// TwinCAT 3 PLC project ShapeMonitor
// ProgramVersion: 3.1.4023.0
// CompilerDefines: VISU_USEWSTRING
// libraries:
//   Tc2_EtherCAT, * (Beckhoff Automation GmbH)
//   Tc2_MDP, * (Beckhoff Automation GmbH)
//   Tc2_ModbusSrv, * (Beckhoff Automation GmbH)
//   Tc2_Standard, * (Beckhoff Automation GmbH)
//   Tc2_System, * (Beckhoff Automation GmbH)
//   Tc2_Utilities, * (Beckhoff Automation GmbH)
//   Tc3_IotBase, * (Beckhoff Automation GmbH)
//   Tc3_IPCDiag, * (Beckhoff Automation GmbH)
//   Tc3_JsonXml, * (Beckhoff Automation GmbH)
//   Tc3_Module, * (Beckhoff Automation GmbH)
//   BASIC,3.31,OSCAT
//   Tc2_SUPS,3.3.8.0,Beckhoff Automation GmbH
//   VisuSymbols,3.5.10.0,System
// project tree:
//   / GlobalTextList.TcGTLO, PlcTask_10ms.TcTTO
//   GVLs/ constGVL.TcGVL, GVL.TcGVL, GVL_outputs.TcGVL
//   HMI/ VisualizationManager.TcVMO (not stored)
//   POUs/FB/ ShapeMonitor.TcPOU
//   POUs/PRG/ Monitoring.TcPOU, Main_T10ms.TcPOU
//   Simulation/ Simulation.TcPOU
// real-time tasks:
//   TASK PlcTask_10ms: cycle T#10ms, priority 20, ADS port 350

CONFIGURATION ShapeMonitor
    RESOURCE PLC ON TwinCAT3
        TASK PlcTask_10ms(INTERVAL := T#10ms, PRIORITY := 20);
        PROGRAM Main_T10ms WITH PlcTask_10ms : Main_T10ms;
    END_RESOURCE
END_CONFIGURATION

// ---- GVLs/constGVL.TcGVL
{attribute 'qualified_only'}
VAR_GLOBAL
	
	//ipHostAddress	: STRING		:= '192.168.1.170';
	ipHostAddress	: STRING		:= '10.1.226.41';
	
	HostPort		: UINT			:= 1883;
	UserName		: STRING		:= 'mqttbroker';
	//UserPassword	: STRING		:= 'LoopEdge.123';
	UserPassword	: STRING		:= 'PLWRO@mqtt';
	
	WorkCenter 		: STRING(30)	:= 'PLPSDWB1';
	LineName 		: STRING(30)	:= 'PSD_WB';
	MachineName01 	: STRING(30)	:= 'WB1';
	MachineTopic_Status01 : STRING	:= 'MachineStatus';
	
	// Config for InfluxDB
	//ActuatorOperTimes_InfluxMeas 	: STRING(50) := 'ActuatorOperTimes';
	VibAccelAnomaly_InfluxMeas 		: STRING(50) := 'VibAccelAnalytics';
	VibVeloAnomaly_InfluxMeas 		: STRING(50) := 'VibVeloAnalytics';
	MachineState_InfluxMeas 		: STRING(50) := 'MachineStatus';
	EdgeDiag_InfluxMeas 			: STRING(50) := 'EdgeGateway';
	FlowSensor_InfluxMeas 			: STRING(50) := 'FlowSensor';
	PressureSensor_InfluxMeas		: STRING(50) := 'PressureSensor';
	PositionSensor_InfluxMeas		: STRING(50) := 'PositionSensor';
	ShapeCorrelation_InfluxMeas		: STRING(50) := 'ShapeCorrelation';
	//TempHumidSensor_InfluxMeas 	: STRING(50) := 'TempHumidSensor';
	//ElectricalData_InfluxMeas		: STRING(50) := 'ElectricalMeasurement';
	
	BF1	:STRING			:= 'BF1';	// przepływ powietrza - zasilanie maszyny
	
	BP1	:STRING			:= 'BP1';	// cisnienie powietrza  - docisk rolek na reduktorem
	BP2	:STRING			:= 'BP2';	// cisnienie powietrza  - odwijanie drutu
	BP3	:STRING			:= 'BP3';	// cisnienie powietrza  - przy enkoderze
	
	// separate vibration sensors 
	BS1 			:STRING			:= 'BS1';		//	wibracje przy kole zębatym - napęd	
	BS2 			:STRING			:= 'BS2';		//	wibracje przy kole zębatym - na obudowie
	BS3				:STRING			:= 'BS3';		// wibracje przy AccuLathe
	
	BG01			:STRING			:='BG01';		// polożenie ciągle ramienia na odwijaku
	BG02			:STRING			:='BG02';		// połozenie binarne ramienia na odwijaku
	
END_VAR

VAR_GLOBAL CONSTANT
	// *******************Global Const ************************
	LeverArmShapeMaxNoSample: UINT := 200;
END_VAR

// ---- GVLs/GVL.TcGVL
{attribute 'qualified_only'}
VAR_GLOBAL
	
(********************* TimeStamp *********************)
	Unix_TimeStamp 			: ULINT;
	
(********************* Machine States *********************)
	AutoMode 				: BOOL;
	ManualMode 				: BOOL;
	MachineProducing		: BOOL;
	DoorGuardSts 			: BOOL;
	ESTOP_NOK				: BOOL;
	
	WireCutSignal			: BOOL;		// command for cutting wire 
	Robot_Error				: BOOL;
	HeatingErrorDepot3		: BOOL;		// heating error on depot 3 (corner)
	HeatingErrorDepot2		: BOOL;		// heating error on depot 2 (middle)
	RobotRunMode			: BOOL;
	WelderRunning			: BOOL;
	WelderReady				: BOOL;
	WelderHeatingOn			: BOOL;
	LifeBeat				: BOOL;		// life bit 1 sec.
	ConnectionOK			: BOOL;		// monitoring of LifeBeat
	FieldbusOK				: BOOL;		// EtherCat communication OK.
	


(**********************************************************)
	ProductOK: DINT;		// amount of finished OK product 
	ProductNOK:	DINT;		// amount of NOK product
	ProductCantNOK:	DINT;	// amount of NOK cant product 
	
	// Data from HMI (PS4800) at WB4
	DataHmi2TwinCat							: ARRAY[1..4] OF DINT;
	
END_VAR

// ---- GVLs/GVL_outputs.TcGVL
{attribute 'qualified_only'}
VAR_GLOBAL
	
	// Data to Allen Bradley over EtherNet/IP
	DataEthNetIP_OUTPUT_DINT0				AT%Q*: DINT;
	DataEthNetIP_OUTPUT_DINT1				AT%Q*: DINT;
END_VAR

// ---- POUs/PRG/Main_T10ms.TcPOU
PROGRAM Main_T10ms
VAR

END_VAR

Simulation();

Monitoring();

END_PROGRAM

// ---- Simulation/Simulation.TcPOU
PROGRAM Simulation
VAR
	BaseValues				:	ARRAY [0..BASE_SHAPE_SAMPLES_NO] OF REAL := [0.1, 0.2, 0.3, 0.5, 0.8, 0.9, 1.0, 1.05, 1.15, 1.25, 1.4, 1.6, 1.8, 2.0, 2.4, 2.8, 3.2, 3.7, 4.1, 4.7, 5.15, 5.6, 6.1, 6.5, 6.95, 7.3, 7.6, 7.9, 8.1, 8.3, 8.4, 3(8.5), 8.4, 8.2, 8.1, 8.0, 7.8, 7.7, 7.5, 7.3, 7.0, 6.98, 6.9, 6.85, 6.9, 6.87, 6.88, 6.85, 6.84, 6.83, 6.84, 6.82, 6.81, 6.82, 6.81, 6.83, 6.8, 6.75, 6.7, 6.65, 6.6, 6.55, 6.5, 6.45, 6.4, 6.35, 6.3, 6.25, 6.2, 6.1, 5.9, 5.8, 5.6, 5.5, 5.32, 5.25, 5.2, 5.0, 4.8, 4.6, 4.4, 4.1, 3.7, 3.4, 3.05, 2.8, 2.6, 2.4, 2.3, 2.1, 1.9, 1.7, 1.5, 1.3, 1.0, 0.7, 0.5, 0.3];
	ValueOffset				:	REAL;
	MeasuredValues			:	ARRAY [0..BASE_SHAPE_SAMPLES_NO] OF REAL;
	Idx						:	UINT;
	SimValue				:	DRAND();
	
	tp01					: 	TP;
	tp02					: 	TP;
	rtShapeStart			:	R_TRIG;
	ftShapeStop				:	F_TRIG;
	ShapeStarted			:	BOOL;
	MeasuredValue			:	REAL;
	SimEnable				:	BOOL;
END_VAR

VAR CONSTANT
	BASE_SHAPE_SAMPLES_NO	: 	UINT:=99;
END_VAR

tp01(IN:=SimEnable AND NOT tp02.Q , PT:=T#1000MS , Q=> , ET=> );
tp02(IN:=NOT tp01.Q , PT:=T#500MS , Q=> , ET=> );

rtShapeStart(CLK:=tp01.Q);
ftShapeStop(CLK:=tp01.Q);

IF rtShapeStart.Q THEN
	ShapeStarted := TRUE;
	Idx := 0;
END_IF

IF ftShapeStop.Q THEN
	ShapeStarted := FALSE;
	MeasuredValue := 0;
END_IF


IF ShapeStarted THEN
	SimValue(Seed:=2);
	ValueOffset := LREAL_TO_REAL(SimValue.Num) - 0.5;
	MeasuredValues[Idx] := BaseValues[Idx] + (0.1 * ValueOffset);
	MeasuredValue := MeasuredValues[Idx];
	Idx := Idx + 1;
	IF Idx > BASE_SHAPE_SAMPLES_NO THEN
		Idx := 0;
		MeasuredValue := 0;
	END_IF
END_IF


//FOR Idx:=0 TO BASE_SHAPE_SAMPLES_NO DO
//	SimValue(Seed:=2);
//	ValueOffset := LREAL_TO_REAL(SimValue.Num) - 0.5;
	
//	MeasuredValues[Idx] := BaseValues[Idx] + (0.2 * ValueOffset);
//END_FOR

END_PROGRAM

// ---- POUs/PRG/Monitoring.TcPOU
PROGRAM Monitoring
VAR	

END_VAR

VAR RETAIN PERSISTENT
	ShapeMonitor01					:	ShapeMonitor;
END_VAR

ShapeMonitor01(
    AnalogIn := Simulation.MeasuredValue,
    TriggerSensor := Simulation.ShapeStarted,
    Enable := TRUE); // ShapeMonitor

END_PROGRAM

// ---- POUs/FB/ShapeMonitor.TcPOU
FUNCTION_BLOCK ShapeMonitor
VAR_INPUT
	AnalogIn											: REAL;
	TriggerSensor										: BOOL;
	Enable												: BOOL;
	Reset												: BOOL;							// reset algorithm
END_VAR
VAR_OUTPUT
	BaseInCalculation									: BOOL;							// base model during calculation
	BaseCompleted										: BOOL;							// model base calculation completed
	SumSquaredError										: REAL;							// SSE - sumed squared error
	Busy												: BOOL;							// shape evaluation in progress 
	Done												: BOOL;							// shape evaluated
END_VAR	

			
VAR
	rtTriggerSensor										: R_TRIG;						// detect rising edge of trigger sensor
	ftTriggerSensor										: F_TRIG;						// detect falling edge of trigger sensor
	rtReset												: R_TRIG;						// detect rising edge of reset signal
	
	State												: (IDLE, TRIGGER_STARTED, TRIGGER_STOPPED );		// state machine
	
	arrShapeSamples										: ARRAY [0..SAMPLES_IN_SHAPE] OF REAL;				// real-time analog samples catched at each PLC scan				
	IdxMeasureSample		   							: UINT;												// index of real-time measured sample 
	
	arrBaseSamples										: ARRAY[0..SHAPES_IN_BASE] OF ARRAY [0..SAMPLES_IN_SHAPE] OF REAL;	// collected real-time signal shapes in base shapes 
	arrNoSamplesInBaseShape								: ARRAY[0..SHAPES_IN_BASE] OF UINT;									// number of samples in each base shape
	arrBase												: ARRAY[0..SAMPLES_IN_SHAPE] OF REAL;								// averaged base shapes array 
	
	arrResult											: ARRAY [0..SAMPLES_IN_SHAPE] OF REAL;								// array with squared diff. between base and incoming new shape
	
	NoBaseShapes										: UINT;																// number of collected shapes in 'base'
	IdxBaseShape										: UINT;																// idx for shape iteration
	IdxSample											: UINT;																// idx for sample iteration
																	
	MaxBaseLength										: UINT;																// max length of shapes in base model
	SampleLength										: UINT;																// length(num of samples) of evaluated shape
	Total												: REAL;																// temporary var
																
END_VAR


VAR CONSTANT
	SHAPES_IN_BASE										: UINT := 10;				// number of shape samples in base
	SAMPLES_IN_SHAPE									: UINT:= 199;				// max number of samples in one shape
END_VAR

// detect rising trigger from reset input	
rtReset(CLK:=Reset , Q=> );	
IF rtReset.Q THEN 
	resetAlgorithm();
END_IF;


IF ENABLE THEN
	
	// detect rising edge of trigger sensor	
	rtTriggerSensor(CLK:=TriggerSensor , Q=> );
	
	// detect falling edge of trigger sensor
	ftTriggerSensor(CLK:=TriggerSensor , Q=> );
	
	CASE State OF
	IDLE:
		// clear array with measured data samples
		MEMSET(ADR(arrShapeSamples), 0, SIZEOF(arrShapeSamples));
		IdxMeasureSample 		:= 0;
		Busy					:= FALSE;	
		Done 					:= FALSE;
		
		IF rtTriggerSensor.Q THEN
			// WatchDog_State_ton.IN := TRUE; //sequence watchdog
			State := TRIGGER_STARTED;
		END_IF
		
	TRIGGER_STARTED:
	// trigger sensor entered start position
		Busy				:= TRUE;	
		Done 				:= FALSE;
		
		// fill the array with incoming measured data
		arrShapeSamples[IdxMeasureSample] := AnalogIn;
		IdxMeasureSample := IdxMeasureSample + 1;
		
		// trigger sensor reached stop position OR max number of samples already collected	
		IF ftTriggerSensor.Q OR IdxMeasureSample > SAMPLES_IN_SHAPE  THEN
			State := TRIGGER_STOPPED;					
		END_IF
		
	TRIGGER_STOPPED:
	// trigger sensor left start position or max no of samples collected
		
		// collect shapes for 'Base' 
		IF NoBaseShapes < SHAPES_IN_BASE  THEN
			BaseInCalculation := TRUE;
			arrBaseSamples[NoBaseShapes] := arrShapeSamples;
			NoBaseShapes := NoBaseShapes + 1;
		
		// shapes for base already collected
		ELSE
			// base calculation not completed yet
			IF NOT BaseCompleted THEN
				
				// find max length of each shape in 'Base'
				FOR IdxBaseShape := 0 TO SHAPES_IN_BASE-1 BY 1 DO
					FOR idxSample := 0 TO SAMPLES_IN_SHAPE BY 1 DO
						IF arrBaseSamples[IdxBaseShape][idxSample] = 0 THEN
							arrNoSamplesInBaseShape[IdxBaseShape] := idxSample-1;
							EXIT;
						END_IF
					END_FOR
				END_FOR
				
				// find max length of all base shapes
				MaxBaseLength 	:= 	0;
				FOR IdxMeasureSample := 0 TO SHAPES_IN_BASE-1 BY 1 DO
					IF arrNoSamplesInBaseShape[IdxMeasureSample] > MaxBaseLength THEN 
						MaxBaseLength:= arrNoSamplesInBaseShape[IdxMeasureSample]; 
					END_IF
				END_FOR
				
				// equalize signal length for all collected base shapes (add last point)
				FOR IdxBaseShape := 0 TO SHAPES_IN_BASE-1 BY 1 DO
					IF arrNoSamplesInBaseShape[IdxBaseShape] <  MaxBaseLength THEN
						FOR IdxSample := arrNoSamplesInBaseShape[IdxBaseShape] TO MaxBaseLength BY 1 DO
							 arrBaseSamples[IdxBaseShape][IdxSample] := arrBaseSamples[IdxBaseShape][ arrNoSamplesInBaseShape[IdxBaseShape]];
						END_FOR
					END_IF
				END_FOR

				// calculate avarage of all samples in BaseSamples -> create one 'Base' array
				FOR IdxSample := 0 TO MaxBaseLength BY 1 DO
					Total := 0;
					FOR  IdxBaseShape := 0 TO SHAPES_IN_BASE-1 BY 1 DO
						Total := Total + arrBaseSamples[IdxBaseShape][IdxSample];
					END_FOR
					arrBase[IdxSample] := Total / (SHAPES_IN_BASE); 
				END_FOR
				
				BaseCompleted	:=	TRUE;
				
			ELSIF BaseCompleted AND
				// ensure that valid number of samples was collected 
				(UINT_TO_REAL(IdxMeasureSample) < 1.1 * UINT_TO_REAL(MaxBaseLength) AND
				 UINT_TO_REAL(IdxMeasureSample) > 0.9 * UINT_TO_REAL(MaxBaseLength) ) THEN
				 
				 BaseInCalculation := FALSE;
				 
				// find length of incoming shape
				FOR IdxSample := 0 TO SAMPLES_IN_SHAPE BY 1 DO
					IF arrShapeSamples[idxSample] = 0 THEN
						SampleLength := idxSample;
						// exit FOR loop when element with value 0 found 
						EXIT;
					END_IF
				END_FOR
				
				// adjust incoming shape length equal to base length by adding last value
				IF SampleLength < MaxBaseLength THEN
					FOR IdxSample := SampleLength TO MaxBaseLength BY 1 DO
						arrShapeSamples[IdxSample] := arrShapeSamples[SampleLength-1];
					END_FOR
				END_IF
				
				// calculate difference between base and measured shape => error and square error value
				FOR IdxSample := 0 TO MaxBaseLength BY 1 DO
					arrResult[idxSample] := LREAL_TO_REAL(EXPT((arrBase[idxSample] - arrShapeSamples[idxSample]),2)) ;
				END_FOR
				
				// calculate sum of squared errors (SSE)
				SumSquaredError := 0;
				FOR IdxSample := 0 TO MaxBaseLength BY 1 DO
					SumSquaredError := SumSquaredError + arrResult[idxSample];
				END_FOR
				
				
			// new samples number is outside of limits -> restart algorithm
			ELSIF BaseCompleted AND (UINT_TO_REAL(IdxMeasureSample) > 1.2 * UINT_TO_REAL(MaxBaseLength)) OR
				  (UINT_TO_REAL(IdxMeasureSample) < 0.8 * UINT_TO_REAL(MaxBaseLength)) THEN
				  // withdraw this shape because too many/too less samples collected
				  resetAlgorithm();
			END_IF
	
		END_IF
		
		
		Busy					:= FALSE;	
		Done 					:= TRUE;
		State					:= IDLE;
		
	END_CASE

ELSE
	;
END_IF

METHOD resetAlgorithm : BOOL
VAR_INPUT
END_VAR
MEMSET(ADR(arrShapeSamples), 0, SIZEOF(arrShapeSamples));
MEMSET(ADR(arrResult), 0, SIZEOF(arrResult));
MEMSET(ADR(arrNoSamplesInBaseShape), 0, SIZEOF(arrNoSamplesInBaseShape));
MEMSET(ADR(arrBase), 0, SIZEOF(arrBase));
MEMSET(ADR(arrBaseSamples), 0, SIZEOF(arrBaseSamples));

IdxMeasureSample				:= 0;
NoBaseShapes					:= 0;

MaxBaseLength 					:= 0;
SampleLength					:= 0;
SumSquaredError					:= 0;

BaseCompleted					:= FALSE;
BaseInCalculation				:= FALSE;
State							:= IDLE;
END_METHOD

END_FUNCTION_BLOCK

// ---- GlobalTextList.TcGTLO
TEXTLIST GlobalTextList
  499 = '%s'
  872 = 'Actuators'
  381 = 'Admin'
  544 = 'Disable'
  871 = 'Electrical'
  199 = 'LAST ACTION'
  325 = 'None'
  130 = 'Operator'
  881 = 'Reset algorithm'
  962 = 'Rst LeverArmCorr'
  957 = 'Rst LeverArmCorrelation'
  966 = 'Rst Vib BS1'
  717 = 'Rst Vib BS2'
  653 = 'Rst Vib BS3'
  413 = 'Service'
  870 = 'Vibration'
END_TEXTLIST
